TYPE TRunCmdTable :
	(
		RCT_None,
		RCT_TakePart,
		RCT_GivePart,
		RCT_Turn,
		RCT_Clean,
		RCT_TurnAndClean
	);
END_TYPE

(* stored: Version 1.1.0.1, ProductVersion 3.1.4022.12
   DUT TRunCmdTable: Id {e243d8dc-50ed-4c58-af36-520f111af5a0} *)
